# EPICS substitutions: PSI/iocGenTime.subs
#GeneralTime not available on EPICS < 3.14.10
file iocGeneralTime.template
{
pattern { IOCNAME }
	{ "$(IOC)"  }
}
